// TIA Portal V20 export
ORGANIZATION_BLOCK "Main"   // OB124, LAD, ProgramCycle
TITLE = "Main Program Sweep (Cycle)"
// stored: Namespace Ely_2, SetENOAutomatically false
   VAR_INPUT
      Initial_Call : Bool;   // Initial call of this OB
      Remanence : Bool;   // =True, if remanent data are available
   END_VAR
BEGIN

REGION Network 1
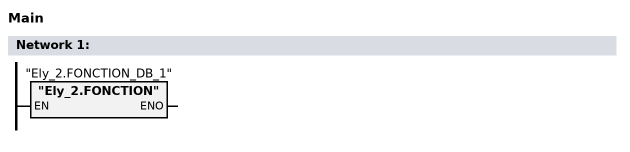
   RUNG wire#powerrail
      "Ely_2.FONCTION_DB_1"()
   END_RUNG
   // the same network as SCL:
   "Ely_2.FONCTION_DB_1"();   // "Ely_2.FONCTION"
END_REGION
END_ORGANIZATION_BLOCK
